PROGRAM LdPrcs
VAR

	ScreenMappingFB: fbV2_ScrMapping;

	fbMainStationProcess_Ld: fbV2_MainStationProcess;
	LdPrcsEN: BOOL;

	bNextBasketAssignIn: BOOL;
	bTimeOptimizedFailedToWrite: BOOL;
	bFailedToWriteHolding: BOOL;
	bA1PnpStep3: BOOL;
	bA1PnpStep3orAbove: BOOL;
	bA1PnpStep1: BOOL;
	bA1PnpStep2: BOOL;
	bMTBScanCompletedFlagHR: BOOL;
	bMTBScanCompletedOnLoadingHR: BOOL;
	LoadingSensorDelayTimer: TON;
	bManualProgramReset: BOOL;

	TrackerStDelayTimer: TON;
	bNextNotAvailableFlag: BOOL;
	bStnTemp1stLimitAlarmTriggered: BOOL;
	bStnConductivityHighAlarmTriggered: BOOL;

	bBasketDetected: BOOL;

	LdStart : BOOL;
	LdReset : BOOL;

	LdProcessFE : F_TRIG;
	LdProcessRE : R_TRIG;
	bCutLdProcessHalt : BOOL;

	bUserDefinePRN_En: BOOL;
	bLdPRNNotMatchFlag: BOOL;
	bLKTTest: BOOL;
	bMinMaxOK: BOOL;
	tLdBasketPickSensorDelayOff: TON;
END_VAR
VAR // added by the converter: edge detectors and wires of the graphical bodies
    _w1, _w2, _w3 : INT;
    _w4 : STRING(INT#4);
    _w5 : BOOL;
END_VAR

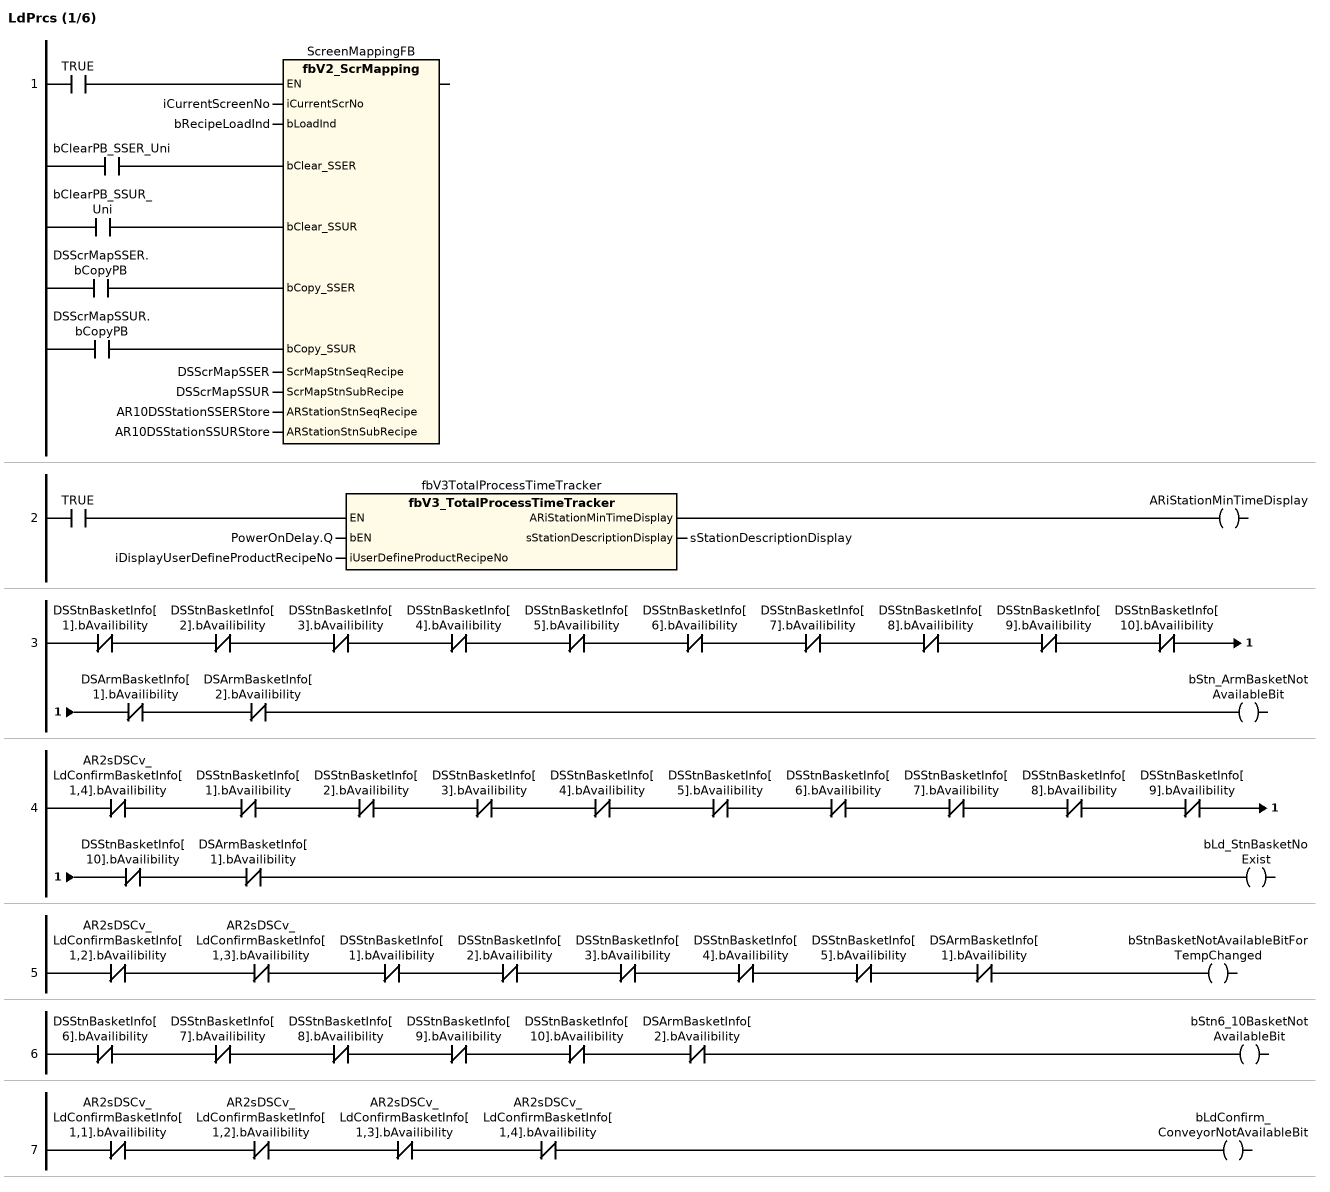
// NETWORK 1
ScreenMappingFB(
    iCurrentScrNo := iCurrentScreenNo,
    bLoadInd := bRecipeLoadInd,
    bClear_SSER := bClearPB_SSER_Uni,
    bClear_SSUR := bClearPB_SSUR_Uni,
    bCopy_SSER := DSScrMapSSER.bCopyPB,
    bCopy_SSUR := DSScrMapSSUR.bCopyPB,
    ScrMapStnSeqRecipe := DSScrMapSSER,
    ScrMapStnSubRecipe := DSScrMapSSUR,
    ARStationStnSeqRecipe := AR10DSStationSSERStore,
    ARStationStnSubRecipe := AR10DSStationSSURStore); // fbV2_ScrMapping

// NETWORK 2
fbV3TotalProcessTimeTracker(
    bEN := PowerOnDelay.Q,
    iUserDefineProductRecipeNo := iDisplayUserDefineProductRecipeNo,
    sStationDescriptionDisplay => sStationDescriptionDisplay); // fbV3_TotalProcessTimeTracker
ARiStationMinTimeDisplay := fbV3TotalProcessTimeTracker.ARiStationMinTimeDisplay;

// NETWORK 3
bStn_ArmBasketNotAvailableBit := NOT DSStnBasketInfo[1].bAvailibility AND NOT DSStnBasketInfo[2].bAvailibility AND NOT DSStnBasketInfo[3].bAvailibility AND NOT DSStnBasketInfo[4].bAvailibility AND NOT DSStnBasketInfo[5].bAvailibility AND NOT DSStnBasketInfo[6].bAvailibility AND NOT DSStnBasketInfo[7].bAvailibility AND NOT DSStnBasketInfo[8].bAvailibility AND NOT DSStnBasketInfo[9].bAvailibility AND NOT DSStnBasketInfo[10].bAvailibility AND NOT DSArmBasketInfo[1].bAvailibility AND NOT DSArmBasketInfo[2].bAvailibility;

// NETWORK 4
bLd_StnBasketNoExist := NOT AR2sDSCv_LdConfirmBasketInfo[1,4].bAvailibility AND NOT DSStnBasketInfo[1].bAvailibility AND NOT DSStnBasketInfo[2].bAvailibility AND NOT DSStnBasketInfo[3].bAvailibility AND NOT DSStnBasketInfo[4].bAvailibility AND NOT DSStnBasketInfo[5].bAvailibility AND NOT DSStnBasketInfo[6].bAvailibility AND NOT DSStnBasketInfo[7].bAvailibility AND NOT DSStnBasketInfo[8].bAvailibility AND NOT DSStnBasketInfo[9].bAvailibility AND NOT DSStnBasketInfo[10].bAvailibility AND NOT DSArmBasketInfo[1].bAvailibility;

// NETWORK 5
bStnBasketNotAvailableBitForTempChanged := (NOT AR2sDSCv_LdConfirmBasketInfo[1,2].bAvailibility AND NOT AR2sDSCv_LdConfirmBasketInfo[1,3].bAvailibility) AND NOT DSStnBasketInfo[1].bAvailibility AND NOT DSStnBasketInfo[2].bAvailibility AND NOT DSStnBasketInfo[3].bAvailibility AND NOT DSStnBasketInfo[4].bAvailibility AND NOT DSStnBasketInfo[5].bAvailibility AND NOT DSArmBasketInfo[1].bAvailibility;

// NETWORK 6
bStn6_10BasketNotAvailableBit := NOT DSStnBasketInfo[6].bAvailibility AND NOT DSStnBasketInfo[7].bAvailibility AND NOT DSStnBasketInfo[8].bAvailibility AND NOT DSStnBasketInfo[9].bAvailibility AND NOT DSStnBasketInfo[10].bAvailibility AND NOT DSArmBasketInfo[2].bAvailibility;

// NETWORK 7
bLdConfirm_ConveyorNotAvailableBit := NOT AR2sDSCv_LdConfirmBasketInfo[1,1].bAvailibility AND NOT AR2sDSCv_LdConfirmBasketInfo[1,2].bAvailibility AND NOT AR2sDSCv_LdConfirmBasketInfo[1,3].bAvailibility AND NOT AR2sDSCv_LdConfirmBasketInfo[1,4].bAvailibility;

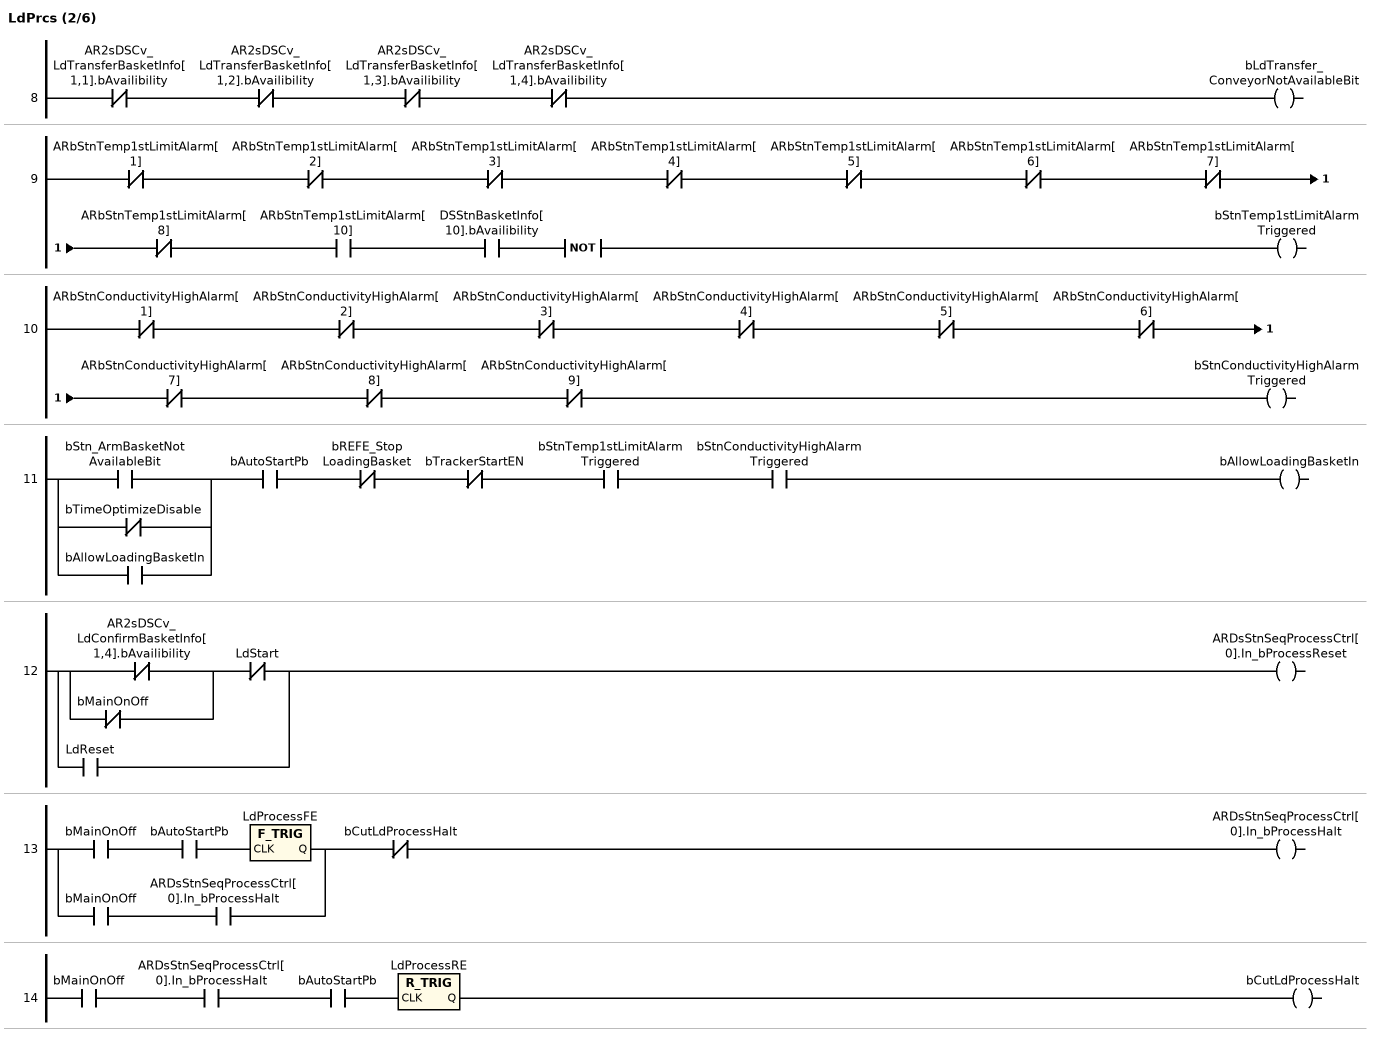
// NETWORK 8
bLdTransfer_ConveyorNotAvailableBit := NOT AR2sDSCv_LdTransferBasketInfo[1,1].bAvailibility AND NOT AR2sDSCv_LdTransferBasketInfo[1,2].bAvailibility AND NOT AR2sDSCv_LdTransferBasketInfo[1,3].bAvailibility AND NOT AR2sDSCv_LdTransferBasketInfo[1,4].bAvailibility;

// NETWORK 9
bStnTemp1stLimitAlarmTriggered := NOT ARbStnTemp1stLimitAlarm[1] AND NOT ARbStnTemp1stLimitAlarm[2] AND NOT ARbStnTemp1stLimitAlarm[3] AND NOT ARbStnTemp1stLimitAlarm[4] AND NOT ARbStnTemp1stLimitAlarm[5] AND NOT ARbStnTemp1stLimitAlarm[6] AND NOT ARbStnTemp1stLimitAlarm[7] AND NOT ARbStnTemp1stLimitAlarm[8] AND NOT (ARbStnTemp1stLimitAlarm[10] AND DSStnBasketInfo[10].bAvailibility);

// NETWORK 10
bStnConductivityHighAlarmTriggered := NOT ARbStnConductivityHighAlarm[1] AND NOT ARbStnConductivityHighAlarm[2] AND NOT ARbStnConductivityHighAlarm[3] AND NOT ARbStnConductivityHighAlarm[4] AND NOT ARbStnConductivityHighAlarm[5] AND NOT ARbStnConductivityHighAlarm[6] AND NOT ARbStnConductivityHighAlarm[7] AND NOT ARbStnConductivityHighAlarm[8] AND NOT ARbStnConductivityHighAlarm[9];

// NETWORK 11
bAllowLoadingBasketIn := (bStn_ArmBasketNotAvailableBit OR NOT bTimeOptimizeDisable OR bAllowLoadingBasketIn) AND bAutoStartPb AND NOT bREFE_StopLoadingBasket AND NOT bTrackerStartEN AND bStnTemp1stLimitAlarmTriggered AND bStnConductivityHighAlarmTriggered;

// NETWORK 12
ARDsStnSeqProcessCtrl[0].In_bProcessReset := (NOT AR2sDSCv_LdConfirmBasketInfo[1,4].bAvailibility OR NOT bMainOnOff) AND NOT LdStart OR LdReset;

// NETWORK 13
LdProcessFE(CLK := bMainOnOff AND bAutoStartPb); // F_TRIG
ARDsStnSeqProcessCtrl[0].In_bProcessHalt := (LdProcessFE.Q OR bMainOnOff AND ARDsStnSeqProcessCtrl[0].In_bProcessHalt) AND NOT bCutLdProcessHalt;

// NETWORK 14
LdProcessRE(CLK := bMainOnOff AND ARDsStnSeqProcessCtrl[0].In_bProcessHalt AND bAutoStartPb); // R_TRIG
bCutLdProcessHalt := LdProcessRE.Q;

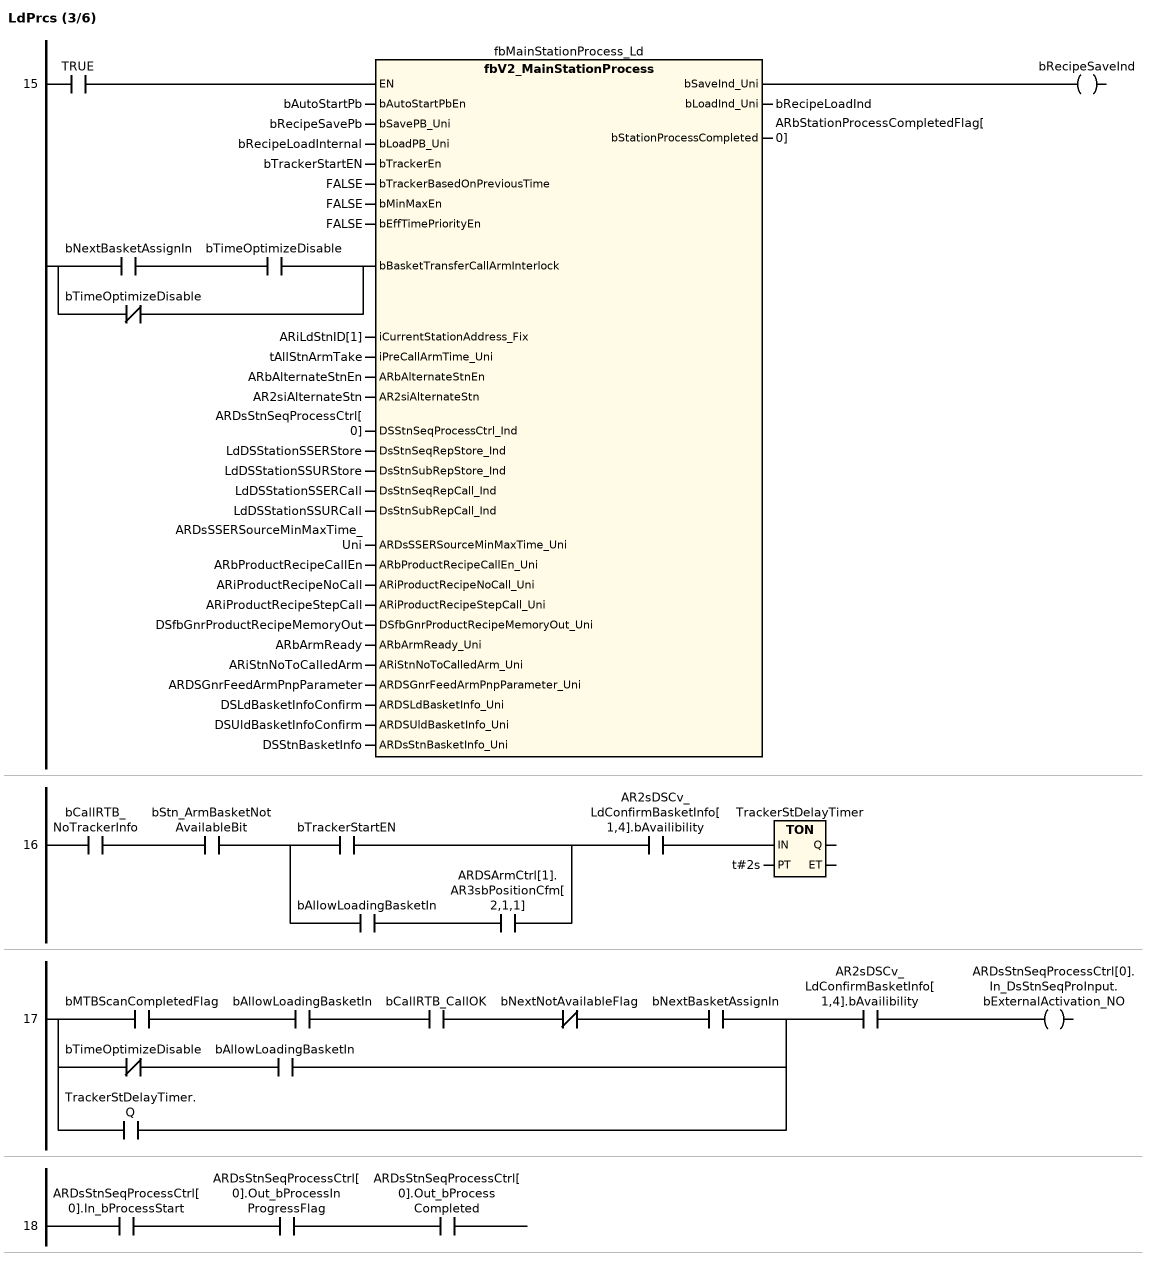
// NETWORK 15
fbMainStationProcess_Ld(
    bAutoStartPbEn := bAutoStartPb,
    bSavePB_Uni := bRecipeSavePb,
    bLoadPB_Uni := bRecipeLoadInternal,
    bTrackerEn := bTrackerStartEN,
    bTrackerBasedOnPreviousTime := FALSE,
    bMinMaxEn := FALSE,
    bEffTimePriorityEn := FALSE,
    bBasketTransferCallArmInterlock := bNextBasketAssignIn AND bTimeOptimizeDisable OR NOT bTimeOptimizeDisable,
    iCurrentStationAddress_Fix := ARiLdStnID[1],
    iPreCallArmTime_Uni := tAllStnArmTake,
    ARbAlternateStnEn := ARbAlternateStnEn,
    AR2siAlternateStn := AR2siAlternateStn,
    DSStnSeqProcessCtrl_Ind := ARDsStnSeqProcessCtrl[0],
    DsStnSeqRepStore_Ind := LdDSStationSSERStore,
    DsStnSubRepStore_Ind := LdDSStationSSURStore,
    DsStnSeqRepCall_Ind := LdDSStationSSERCall,
    DsStnSubRepCall_Ind := LdDSStationSSURCall,
    ARDsSSERSourceMinMaxTime_Uni := ARDsSSERSourceMinMaxTime_Uni,
    ARbProductRecipeCallEn_Uni := ARbProductRecipeCallEn,
    ARiProductRecipeNoCall_Uni := ARiProductRecipeNoCall,
    ARiProductRecipeStepCall_Uni := ARiProductRecipeStepCall,
    DSfbGnrProductRecipeMemoryOut_Uni := DSfbGnrProductRecipeMemoryOut,
    ARbArmReady_Uni := ARbArmReady,
    ARiStnNoToCalledArm_Uni := ARiStnNoToCalledArm,
    ARDSGnrFeedArmPnpParameter_Uni := ARDSGnrFeedArmPnpParameter,
    ARDSLdBasketInfo_Uni := DSLdBasketInfoConfirm,
    ARDSUldBasketInfo_Uni := DSUldBasketInfoConfirm,
    ARDsStnBasketInfo_Uni := DSStnBasketInfo,
    bLoadInd_Uni => bRecipeLoadInd,
    bStationProcessCompleted => ARbStationProcessCompletedFlag[0]); // fbV2_MainStationProcess
bRecipeSaveInd := fbMainStationProcess_Ld.bSaveInd_Uni;

// NETWORK 16
TrackerStDelayTimer(IN := (bCallRTB_NoTrackerInfo AND bStn_ArmBasketNotAvailableBit AND (bTrackerStartEN OR bAllowLoadingBasketIn AND ARDSArmCtrl[1].AR3sbPositionCfm[2,1,1])) AND AR2sDSCv_LdConfirmBasketInfo[1,4].bAvailibility, PT := t#2s); // TON

// NETWORK 17
ARDsStnSeqProcessCtrl[0].In_DsStnSeqProInput.bExternalActivation_NO := (bMTBScanCompletedFlag AND bAllowLoadingBasketIn AND bCallRTB_CallOK AND NOT bNextNotAvailableFlag AND bNextBasketAssignIn OR NOT bTimeOptimizeDisable AND bAllowLoadingBasketIn OR TrackerStDelayTimer.Q) AND AR2sDSCv_LdConfirmBasketInfo[1,4].bAvailibility;

// NETWORK 18
(* ARDsStnSeqProcessCtrl[0].In_bProcessStart AND ARDsStnSeqProcessCtrl[0].Out_bProcessInProgressFlag AND ARDsStnSeqProcessCtrl[0].Out_bProcessCompleted; result not used *)

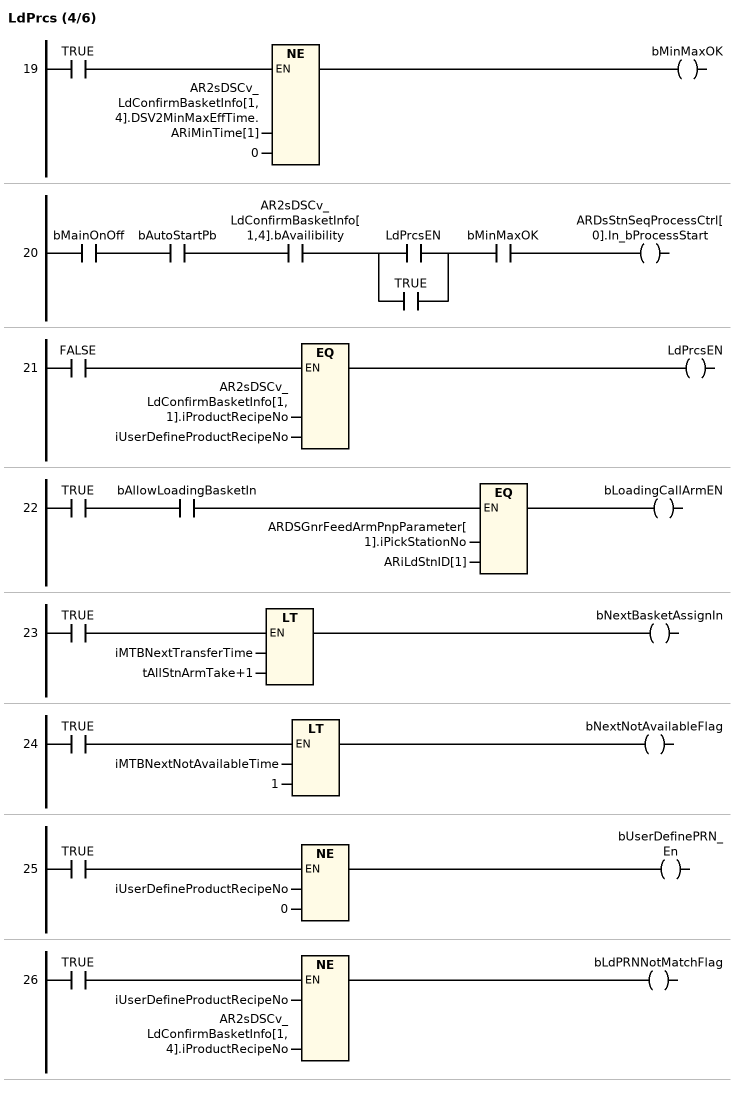
// NETWORK 19
bMinMaxOK := AR2sDSCv_LdConfirmBasketInfo[1,4].DSV2MinMaxEffTime.ARiMinTime[1] <> 0;

// NETWORK 20
ARDsStnSeqProcessCtrl[0].In_bProcessStart := (bMainOnOff AND bAutoStartPb AND AR2sDSCv_LdConfirmBasketInfo[1,4].bAvailibility AND (LdPrcsEN OR TRUE)) AND bMinMaxOK;

// NETWORK 21
LdPrcsEN := FALSE AND AR2sDSCv_LdConfirmBasketInfo[1,1].iProductRecipeNo = iUserDefineProductRecipeNo;

// NETWORK 22
bLoadingCallArmEN := TRUE AND bAllowLoadingBasketIn AND ARDSGnrFeedArmPnpParameter[1].iPickStationNo = ARiLdStnID[1];

// NETWORK 23
bNextBasketAssignIn := iMTBNextTransferTime < (tAllStnArmTake+1);

// NETWORK 24
bNextNotAvailableFlag := iMTBNextNotAvailableTime < 1;

// NETWORK 25
bUserDefinePRN_En := iUserDefineProductRecipeNo <> 0;

// NETWORK 26
bLdPRNNotMatchFlag := iUserDefineProductRecipeNo <> AR2sDSCv_LdConfirmBasketInfo[1,4].iProductRecipeNo;

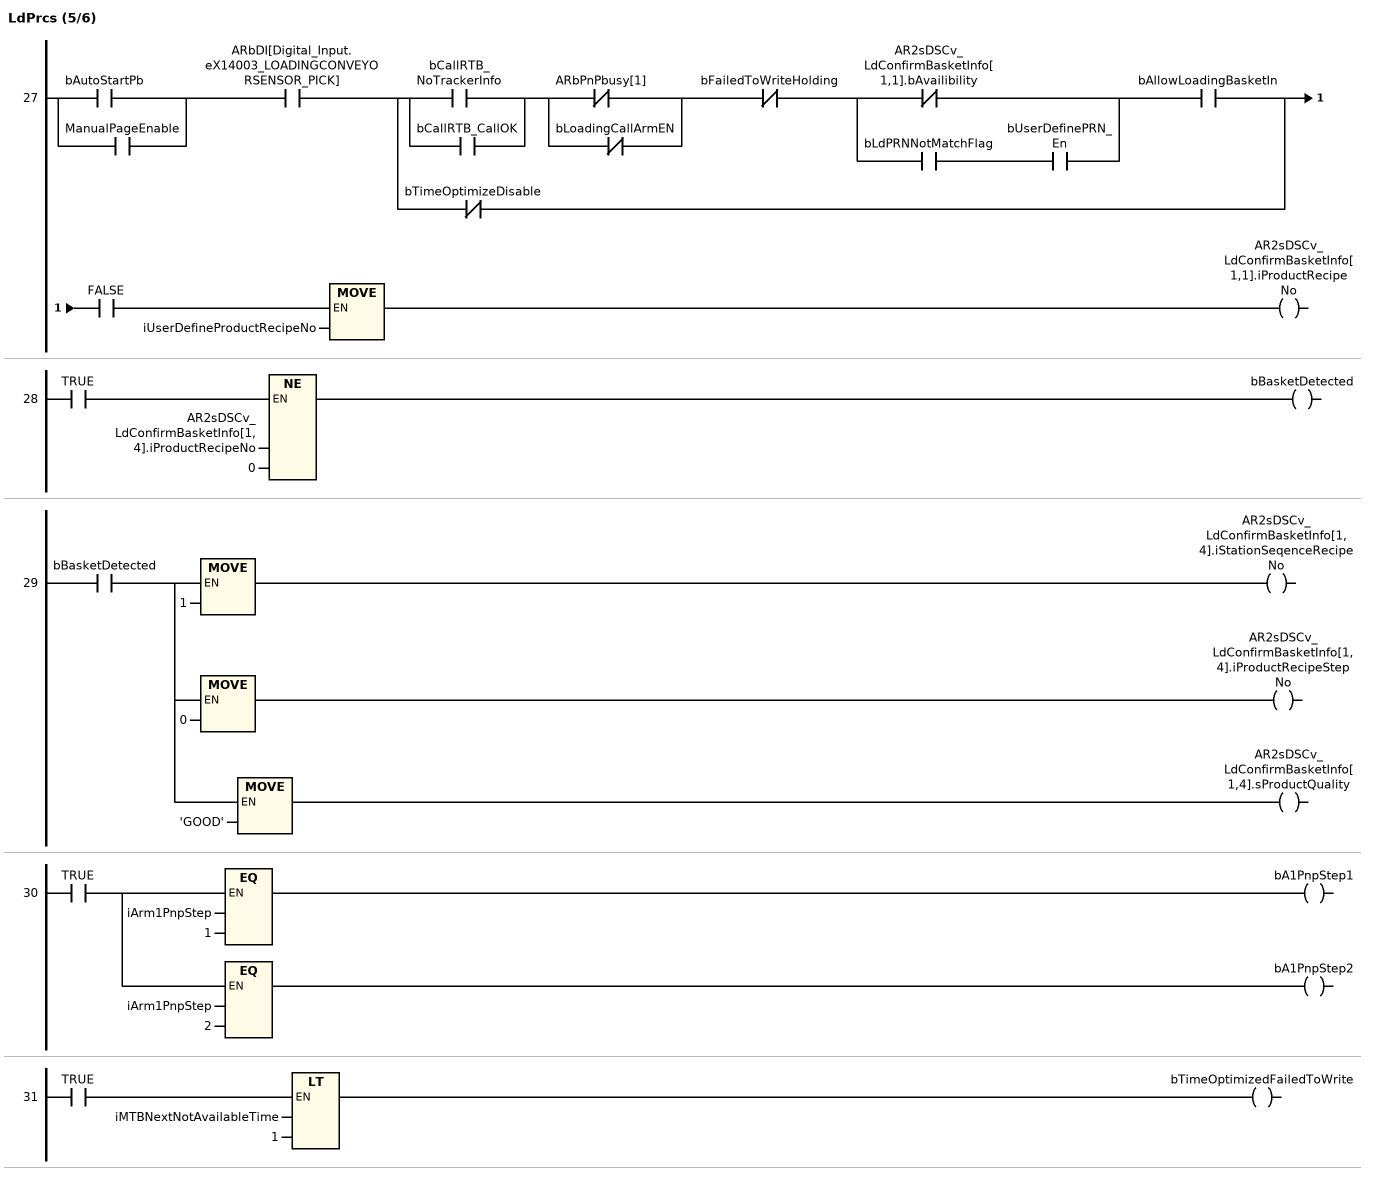
// NETWORK 27
IF ((bAutoStartPb OR ManualPageEnable) AND ARbDI[Digital_Input.eX14003_LOADINGCONVEYORSENSOR_PICK] AND ((((bCallRTB_NoTrackerInfo OR bCallRTB_CallOK) AND (NOT ARbPnPbusy[1] OR NOT bLoadingCallArmEN)) AND NOT bFailedToWriteHolding AND (NOT AR2sDSCv_LdConfirmBasketInfo[1,1].bAvailibility OR bLdPRNNotMatchFlag AND bUserDefinePRN_En)) AND bAllowLoadingBasketIn OR NOT bTimeOptimizeDisable)) AND FALSE THEN
    _w1 := iUserDefineProductRecipeNo;
END_IF
AR2sDSCv_LdConfirmBasketInfo[1,1].iProductRecipeNo := _w1;

// NETWORK 28
bBasketDetected := AR2sDSCv_LdConfirmBasketInfo[1,4].iProductRecipeNo <> 0;

// NETWORK 29
IF bBasketDetected THEN _w2 := 1; END_IF
AR2sDSCv_LdConfirmBasketInfo[1,4].iStationSeqenceRecipeNo := _w2;
IF bBasketDetected THEN _w3 := 0; END_IF
AR2sDSCv_LdConfirmBasketInfo[1,4].iProductRecipeStepNo := _w3;
IF bBasketDetected THEN _w4 := 'GOOD'; END_IF
AR2sDSCv_LdConfirmBasketInfo[1,4].sProductQuality := _w4;

// NETWORK 30
bA1PnpStep1 := iArm1PnpStep = 1;
bA1PnpStep2 := iArm1PnpStep = 2;

// NETWORK 31
bTimeOptimizedFailedToWrite := iMTBNextNotAvailableTime < 1;

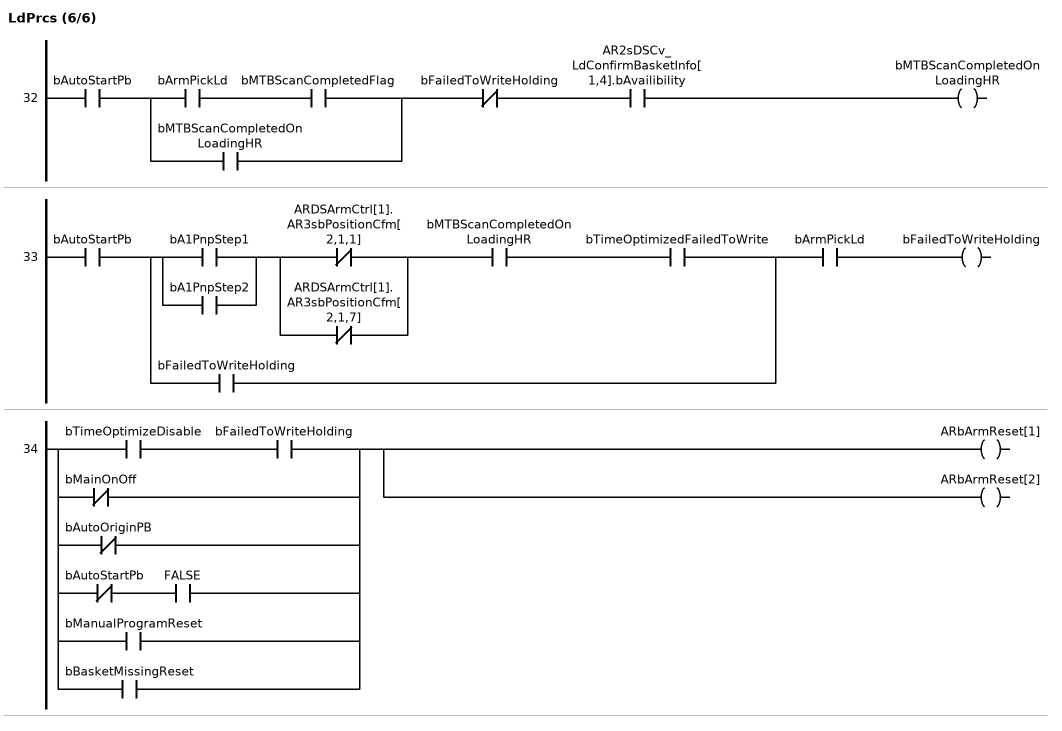
// NETWORK 32
bMTBScanCompletedOnLoadingHR := (bAutoStartPb AND (bArmPickLd AND bMTBScanCompletedFlag OR bMTBScanCompletedOnLoadingHR)) AND NOT bFailedToWriteHolding AND AR2sDSCv_LdConfirmBasketInfo[1,4].bAvailibility;

// NETWORK 33
bFailedToWriteHolding := (bAutoStartPb AND (((bA1PnpStep1 OR bA1PnpStep2) AND (NOT ARDSArmCtrl[1].AR3sbPositionCfm[2,1,1] OR NOT ARDSArmCtrl[1].AR3sbPositionCfm[2,1,7])) AND bMTBScanCompletedOnLoadingHR AND bTimeOptimizedFailedToWrite OR bFailedToWriteHolding)) AND bArmPickLd;

// NETWORK 34
_w5 := bTimeOptimizeDisable AND bFailedToWriteHolding OR NOT bMainOnOff OR NOT bAutoOriginPB OR NOT bAutoStartPb AND FALSE OR bManualProgramReset OR bBasketMissingReset;
ARbArmReset[1] := _w5;
ARbArmReset[2] := _w5;

ACTION NoBasketDetected:
IF NOT bBasketDetected THEN
	AR2sDSCv_LdConfirmBasketInfo[1,4].iProductRecipeStepNo:=0;
	AR2sDSCv_LdConfirmBasketInfo[1,4].iStationSeqenceRecipeNo:=0;
END_IF
END_ACTION

END_PROGRAM

(* stored: Version 1.1.0.1, ProductVersion 3.1.4024.12
   POU LdPrcs: Id {7518fc51-3e01-4537-8eb8-5da333556a85}, SpecialFunc None
   Action NoBasketDetected: Id {684b713c-fdba-45b2-b983-517ba35ca3a7} *)
